{attribute addProperty BoxType "EL3314-0010-0016"}
{attribute addProperty Id "TC_Inputs_ChannelAT %I*ARRAY[0..3] OF TC_Inputs_Channel_842FAF6F50062.50WcStateAT %I*WcState_98A4DF7520.250InfoDataAT %I*InfoData_BC63D37F80100"}
{attribute addProperty CRC "4098794786"}
{attribute addProperty SizeInBites "582"}
{attribute addProperty SizeInBytes "72.75"}
TYPE EL3314_FE14BA1D :
STRUCT
	{attribute addProperty Name "TC_Inputs_Channel"}
	TC_Inputs_Channel : ARRAY[0..3] OF TC_Inputs_Channel_842FAF6F;
	{attribute addProperty Name "WcState"}
	WcState : WcState_98A4DF75;
	{attribute addProperty Name "InfoData"}
	InfoData : InfoData_BC63D37F;
END_STRUCT
END_TYPE

(* stored: Version 1.2.0.0, ProductVersion 3.1.4024.9
   DUT EL3314_FE14BA1D: Id {86e7ab4a-8e56-4e4b-ad10-62047c02dca7} *)
